PROGRAM Vision_GUI_Control
VAR


	
END_VAR

END_PROGRAM

(* stored: Version 1.1.0.1, ProductVersion 3.1.4024.12
   POU Vision_GUI_Control: Id {87634a6b-c49e-421c-811e-918241457a4d}, SpecialFunc None *)
